TYPE ST_DeviceIO :
STRUCT
	stIn 	AT%I* : ST_DeviceIn;
	stOut	AT%Q* : ST_DeviceOut;
END_STRUCT
END_TYPE

(* stored: Version 1.1.0.1, ProductVersion 3.1.4020.12
   DUT ST_DeviceIO: Id {741dfcf9-fe2b-4a9a-a51b-35e9cbed7eb5} *)
